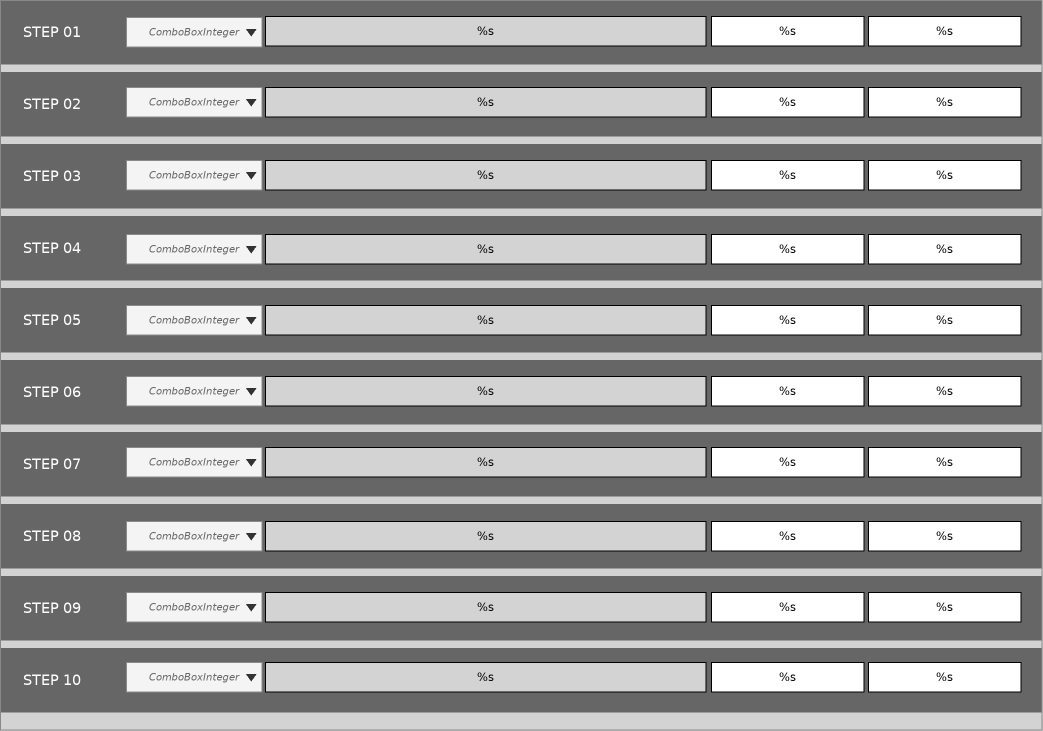
VISUALIZATION Popup_RecipeSSER  // 1043x731
    Rectangle (0,0 1043x731)
    RoundedRectangle (0,360 1042x64)
    Label (20,380 103x24), "STEP 06"
    RoundedRectangle (0,432 1042x64)
    Label (20,452 103x24), "STEP 07"
    RoundedRectangle (0,504 1042x64)
    Label (20,524 103x24), "STEP 08"
    RoundedRectangle (0,576 1042x64)
    Label (20,596 103x24), "STEP 09"
    RoundedRectangle (0,648 1042x64)
    Label (20,668 103x24), "STEP 10"
    RoundedRectangle (0,0 1042x64)
    Label (20,20 103x24), "STEP 01"
    RoundedRectangle (0,72 1042x64)
    Label (20,92 103x24), "STEP 02"
    RoundedRectangle (0,144 1042x64)
    Label (20,164 103x24), "STEP 03"
    RoundedRectangle (0,216 1042x64)
    Label (20,236 103x24), "STEP 04"
    RoundedRectangle (0,288 1042x64)
    Label (20,308 103x24), "STEP 05"
    ComboBoxInteger (126,376 136x30), variable: DSScrMapSSER.DsStationSequenceRecipeMemory.AR10iStationSubProNo[6], text list: 'TextList_1_20'
    RoundedRectangle (265,376 441x30), "%s", text variable: ARsHMIDisplaySSURDescription[6]
    ComboBoxInteger (126,447 136x30), variable: DSScrMapSSER.DsStationSequenceRecipeMemory.AR10iStationSubProNo[7], text list: 'TextList_1_20'
    RoundedRectangle (265,447 441x30), "%s", text variable: ARsHMIDisplaySSURDescription[7]
    ComboBoxInteger (126,521 136x30), variable: DSScrMapSSER.DsStationSequenceRecipeMemory.AR10iStationSubProNo[8], text list: 'TextList_1_20'
    RoundedRectangle (265,521 441x30), "%s", text variable: ARsHMIDisplaySSURDescription[8]
    ComboBoxInteger (126,592 136x30), variable: DSScrMapSSER.DsStationSequenceRecipeMemory.AR10iStationSubProNo[9], text list: 'TextList_1_20'
    RoundedRectangle (265,592 441x30), "%s", text variable: ARsHMIDisplaySSURDescription[9]
    ComboBoxInteger (126,662 136x30), variable: DSScrMapSSER.DsStationSequenceRecipeMemory.AR10iStationSubProNo[10], text list: 'TextList_1_20'
    RoundedRectangle (265,662 441x30), "%s", text variable: ARsHMIDisplaySSURDescription[10]
    ComboBoxInteger (126,17 136x30), variable: DSScrMapSSER.DsStationSequenceRecipeMemory.AR10iStationSubProNo[1], text list: 'TextList_1_20'
    RoundedRectangle (265,16 441x30), "%s", text variable: ARsHMIDisplaySSURDescription[1]
    ComboBoxInteger (126,87 136x30), variable: DSScrMapSSER.DsStationSequenceRecipeMemory.AR10iStationSubProNo[2], text list: 'TextList_1_20'
    RoundedRectangle (265,87 441x30), "%s", text variable: ARsHMIDisplaySSURDescription[2]
    ComboBoxInteger (126,160 136x30), variable: DSScrMapSSER.DsStationSequenceRecipeMemory.AR10iStationSubProNo[3], text list: 'TextList_1_20'
        p1601986498: ''
    RoundedRectangle (265,160 441x30), "%s", text variable: ARsHMIDisplaySSURDescription[3]
    ComboBoxInteger (126,234 136x30), variable: DSScrMapSSER.DsStationSequenceRecipeMemory.AR10iStationSubProNo[4], text list: 'TextList_1_20'
    RoundedRectangle (265,234 441x30), "%s", text variable: ARsHMIDisplaySSURDescription[4]
    ComboBoxInteger (126,305 136x30), variable: DSScrMapSSER.DsStationSequenceRecipeMemory.AR10iStationSubProNo[5], text list: 'TextList_1_20'
    RoundedRectangle (265,305 441x30), "%s", text variable: ARsHMIDisplaySSURDescription[5]
    RoundedRectangle (711,16 153x30), "%s", text variable: DSScrMapSSER.DsStationSequenceRecipeMemory.AR10iCycle[1]
        OnMouseDown: write the text variable via VisuDialogs.Numpad, min 1, max 99
    RoundedRectangle (868,16 153x30), "%s", text variable: DSScrMapSSER.DsStationSequenceRecipeMemory.AR10iRepeatFromStepNo[1]
        OnMouseDown: write the text variable via VisuDialogs.Numpad, min 1, max 10
    RoundedRectangle (711,87 153x30), "%s", text variable: DSScrMapSSER.DsStationSequenceRecipeMemory.AR10iCycle[2]
        OnMouseDown: write the text variable via VisuDialogs.Numpad, min 1, max 99
    RoundedRectangle (868,87 153x30), "%s", text variable: DSScrMapSSER.DsStationSequenceRecipeMemory.AR10iRepeatFromStepNo[2]
        OnMouseDown: write the text variable via VisuDialogs.Numpad, min 1, max 10
    RoundedRectangle (711,160 153x30), "%s", text variable: DSScrMapSSER.DsStationSequenceRecipeMemory.AR10iCycle[3]
        OnMouseDown: write the text variable via VisuDialogs.Numpad, min 1, max 99
    RoundedRectangle (868,160 153x30), "%s", text variable: DSScrMapSSER.DsStationSequenceRecipeMemory.AR10iRepeatFromStepNo[3]
        OnMouseDown: write the text variable via VisuDialogs.Numpad, min 1, max 10
    RoundedRectangle (711,234 153x30), "%s", text variable: DSScrMapSSER.DsStationSequenceRecipeMemory.AR10iCycle[4]
        OnMouseDown: write the text variable via VisuDialogs.Numpad, min 1, max 99
    RoundedRectangle (868,234 153x30), "%s", text variable: DSScrMapSSER.DsStationSequenceRecipeMemory.AR10iRepeatFromStepNo[4]
        OnMouseDown: write the text variable via VisuDialogs.Numpad, min 1, max 10
    RoundedRectangle (711,305 153x30), "%s", text variable: DSScrMapSSER.DsStationSequenceRecipeMemory.AR10iCycle[5]
        OnMouseDown: write the text variable via VisuDialogs.Numpad, min 1, max 99
    RoundedRectangle (868,305 153x30), "%s", text variable: DSScrMapSSER.DsStationSequenceRecipeMemory.AR10iRepeatFromStepNo[5]
        OnMouseDown: write the text variable via VisuDialogs.Numpad, min 1, max 10
    RoundedRectangle (711,376 153x30), "%s", text variable: DSScrMapSSER.DsStationSequenceRecipeMemory.AR10iCycle[6]
        OnMouseDown: write the text variable via VisuDialogs.Numpad, min 1, max 99
    RoundedRectangle (868,376 153x30), "%s", text variable: DSScrMapSSER.DsStationSequenceRecipeMemory.AR10iRepeatFromStepNo[6]
        OnMouseDown: write the text variable via VisuDialogs.Numpad, min 1, max 10
    RoundedRectangle (711,447 153x30), "%s", text variable: DSScrMapSSER.DsStationSequenceRecipeMemory.AR10iCycle[7]
        OnMouseDown: write the text variable via VisuDialogs.Numpad, min 1, max 99
    RoundedRectangle (868,447 153x30), "%s", text variable: DSScrMapSSER.DsStationSequenceRecipeMemory.AR10iRepeatFromStepNo[7]
        OnMouseDown: write the text variable via VisuDialogs.Numpad, min 1, max 10
    RoundedRectangle (711,521 153x30), "%s", text variable: DSScrMapSSER.DsStationSequenceRecipeMemory.AR10iCycle[8]
        OnMouseDown: write the text variable via VisuDialogs.Numpad, min 1, max 99
    RoundedRectangle (868,521 153x30), "%s", text variable: DSScrMapSSER.DsStationSequenceRecipeMemory.AR10iRepeatFromStepNo[8]
        OnMouseDown: write the text variable via VisuDialogs.Numpad, min 1, max 10
    RoundedRectangle (711,592 153x30), "%s", text variable: DSScrMapSSER.DsStationSequenceRecipeMemory.AR10iCycle[9]
        OnMouseDown: write the text variable via VisuDialogs.Numpad, min 1, max 99
    RoundedRectangle (868,592 153x30), "%s", text variable: DSScrMapSSER.DsStationSequenceRecipeMemory.AR10iRepeatFromStepNo[9]
        OnMouseDown: write the text variable via VisuDialogs.Numpad, min 1, max 10
    RoundedRectangle (711,662 153x30), "%s", text variable: DSScrMapSSER.DsStationSequenceRecipeMemory.AR10iCycle[10]
        OnMouseDown: write the text variable via VisuDialogs.Numpad, min 1, max 99
    RoundedRectangle (868,662 153x30), "%s", text variable: DSScrMapSSER.DsStationSequenceRecipeMemory.AR10iRepeatFromStepNo[10]
        OnMouseDown: write the text variable via VisuDialogs.Numpad, min 1, max 10
END_VISUALIZATION

(* stored: Version 1.1.0.1, ProductVersion 3.1.4024.12
   Visu Popup_RecipeSSER: Id {ca77f390-c624-45ef-a8db-de1ba050a11e} *)
